{attribute 'qualified_only'}
{attribute 'strict'}
TYPE E_DataType :
(
	eDataType_None := 0,
	eDataType_bool,
	eDataType_int,
	eDataType_lreal,
	eDataType_wstring,
	eDataType_time_ms,
	eDataType_time_s,
	eDataType_time_m,
	eDataType_time_h,
	
	eDataType_Max
);
END_TYPE

(* stored: Version 1.1.0.1
   EnumerationTextList E_DataType: Id {e0b66050-ff2c-4a62-8ba8-40a71306ddcc} *)
